Staubli VAL3: onF4Event.pgx

program onF4Event()
begin
   // look if the bButton is enable
  if bButton[3]
    //
  endIf
end
